// TIA Portal V18 export
DATA_BLOCK "blinker_LEDDESK"   // DB25
VERSION : 0.1
// stored: AutoNumber true, DBAccessibleFromOPCUA true, InstanceOfName BLINKER, InstanceOfType FB
"BLINKER"
   // VAR_INPUT
   //    BLINK_NOW : Bool;
   //    ON_t : Time;
   //    OFF_t : Time;
   // END_VAR
   // VAR_OUTPUT
   //    yToBlink : Bool;
   // END_VAR
   // VAR
   //    tON_DB { S7_SetPoint := 'True'} : TON_TIME;
   //    tOFF_DB { S7_SetPoint := 'True'} : TON_TIME;
   //    off_mem { S7_SetPoint := 'True'} : Bool;
   // END_VAR
BEGIN
END_DATA_BLOCK
